Yaskawa INFORM job: SRCH-TEST.JBI

/JOB
//NAME SRCH-TEST
///FOLDERNAME OTHER
//POS
///NPOS 2,2,0,0,0,0
///TOOL 0
///POSTYPE ROBOT
///RECTAN
///RCONF 1,0,1,0,0,0,0,0,0,0,0,0,0,0,0,0,0,0,0,0,0,0,0,0
C00000=641.588,-641.596,290.672,6.7809,-24.6454,-92.9821
C00001=667.755,-641.661,293.502,6.7836,-24.6449,-92.9851
///RCONF 0,0,0,0,0,0,0,0,0,0,0,0,0,0,0,0,0,0,0,0,0,0,0,0
BC00000=0.046
BC00001=0.046
//INST
///DATE 2024/02/28 12:57
///ATTR SC,RW,RJ
////FRAME ROBOT
///GROUP1 RB1,BS1
///LVARS 1,0,0,0,0,0,0,0
NOP
MOVL C00000 BC00000 V=11.0
MOVL C00001 BC00001 V=11.0 SRCH RIN#(1)=ON DIS=0.1
GETS LB000 $B002
IFTHENEXP LB000=0
	 PAUSE
	'FAIL
	 PAUSE
ENDIF
END
